TYPE ST_ProcessStatus :
STRUCT
    eMode                      : E_MainMode;
    eState                     : E_MainState;
    eOperation                 : E_MainOperation;
    eAutoPhase                 : E_AutoPhase;
	
	eAutoRouteReq				: E_Route;

    bAutoCycleActive           : BOOL;
    bManualCycleActive         : BOOL;

    bReadyToStart              : BOOL;
    bInPause                   : BOOL;
    bInFault                   : BOOL;

    iStatusCode                : INT;
END_STRUCT
END_TYPE

(* stored: Version 1.1.0.1, ProductVersion 3.1.4024.16
   DUT ST_ProcessStatus: Id {c1497a6c-4050-47d9-9940-fcf57961c2d1} *)
